// Mitsubishi GX Developer project: PLC_PCO520L2   PLC: Q06UDEH   Door Open Auto Flow

PROGRAM AT_DOAT
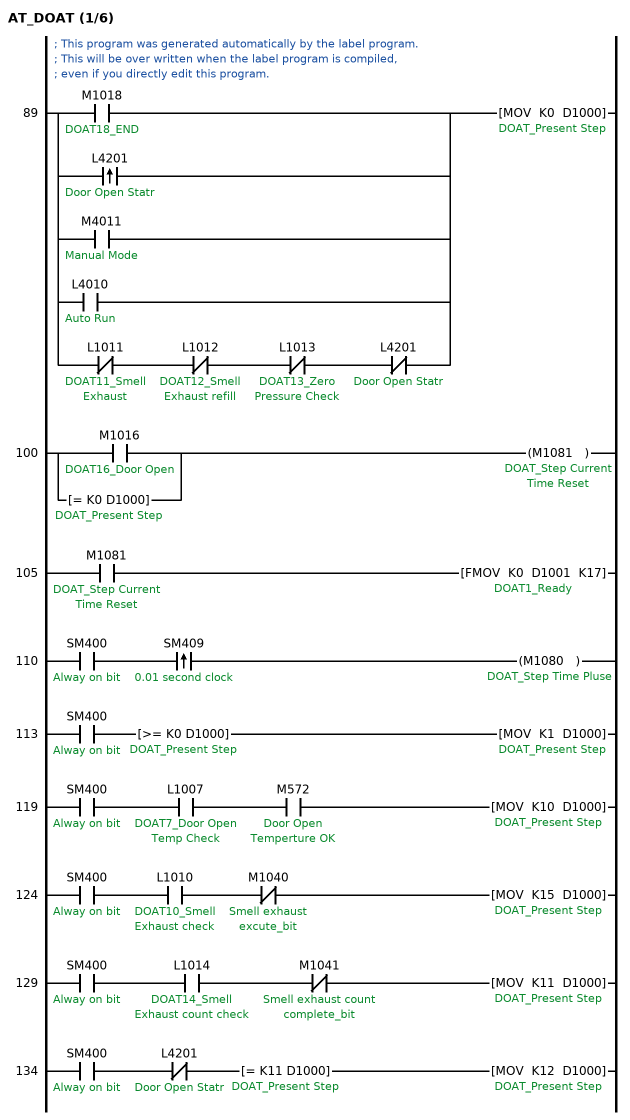
; This program was generated automatically by the label program.
; This will be over written when the label program is compiled,
; even if you directly edit this program.
89    LD      M1018  ; DOAT18_END
      ORP     L4201  ; Door Open Statr
      OR      M4011  ; Manual Mode
      OR      L4010  ; Auto Run
      LDI     L1011  ; DOAT11_Smell Exhaust
      ANI     L1012  ; DOAT12_Smell Exhaust refill
      ANI     L1013  ; DOAT13_Zero Pressure Check
      ANI     L4201  ; Door Open Statr
      ORB
      MOV     K0 D1000  ; DOAT_Present Step
100   LD      M1016  ; DOAT16_Door Open
      OR=     K0 D1000  ; DOAT_Present Step
      OUT     M1081  ; DOAT_Step Current Time Reset
105   LD      M1081  ; DOAT_Step Current Time Reset
      FMOV    K0 D1001 K17  ; DOAT1_Ready
110   LD      SM400  ; Alway on bit
      ANDP    SM409  ; 0.01 second clock
      OUT     M1080  ; DOAT_Step Time Pluse
113   LD      SM400  ; Alway on bit
      AND>=   K0 D1000  ; DOAT_Present Step
      MOV     K1 D1000
119   LD      SM400  ; Alway on bit
      AND     L1007  ; DOAT7_Door Open Temp Check
      AND     M572  ; Door Open Temperture OK
      MOV     K10 D1000
124   LD      SM400  ; Alway on bit
      AND     L1010  ; DOAT10_Smell Exhaust check
      ANI     M1040  ; Smell exhaust excute_bit
      MOV     K15 D1000
129   LD      SM400  ; Alway on bit
      AND     L1014  ; DOAT14_Smell Exhaust count check
      ANI     M1041  ; Smell exhaust count complete_bit
      MOV     K11 D1000
134   LD      SM400  ; Alway on bit
      ANI     L4201  ; Door Open Statr
      AND=    K11 D1000  ; DOAT_Present Step
      MOV     K12 D1000
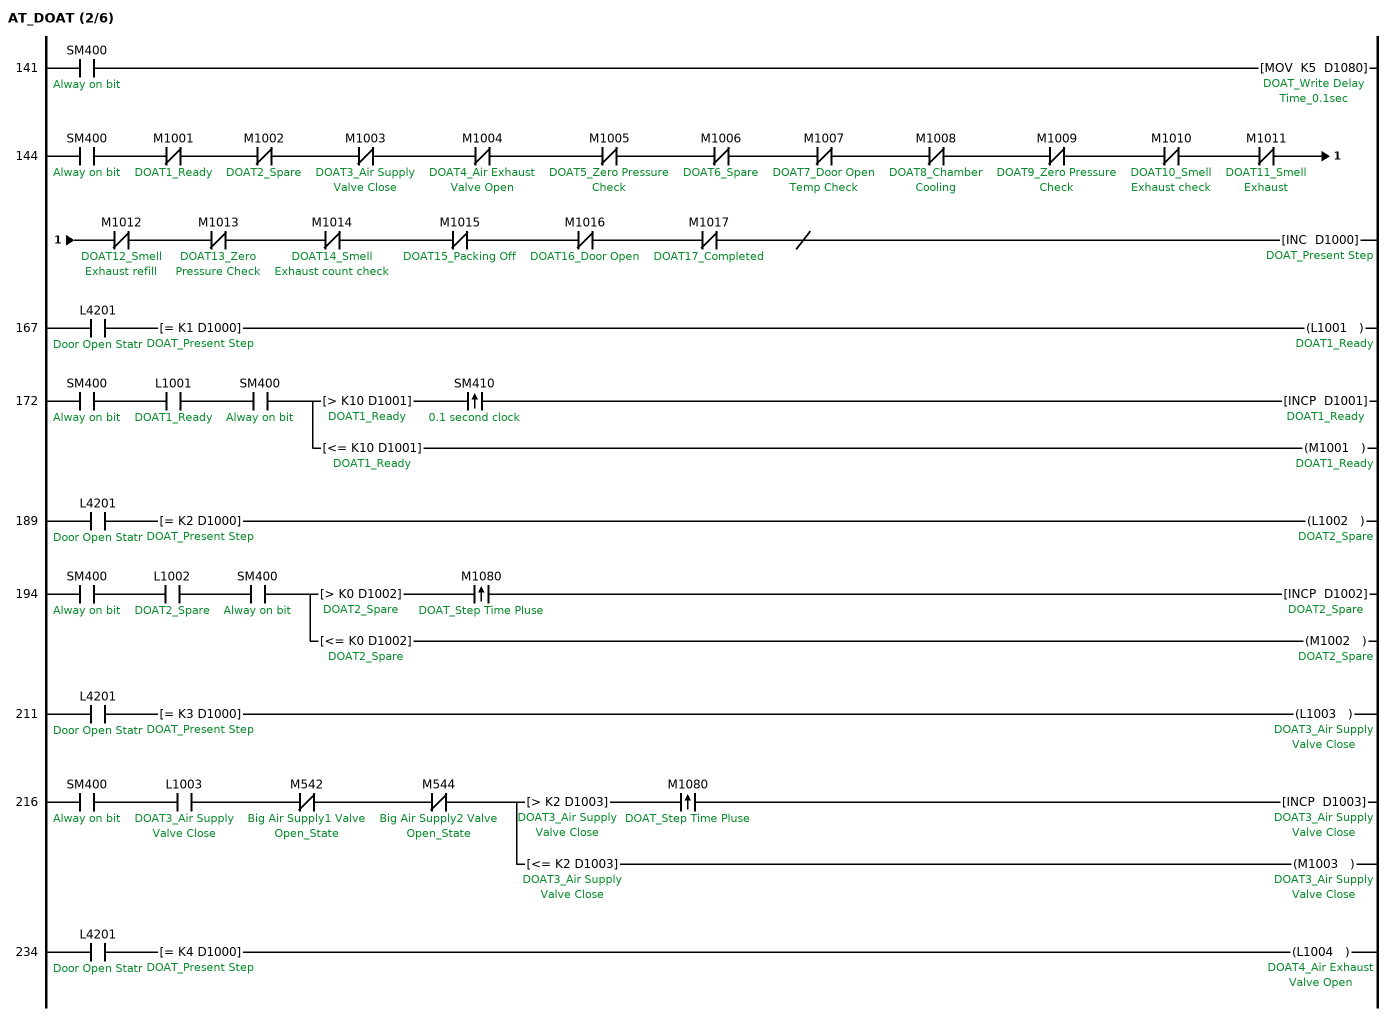
141   LD      SM400  ; Alway on bit
      MOV     K5 D1080  ; DOAT_Write Delay Time_0.1sec
144   LD      SM400  ; Alway on bit
      ANI     M1001  ; DOAT1_Ready
      ANI     M1002  ; DOAT2_Spare
      ANI     M1003  ; DOAT3_Air Supply Valve Close
      ANI     M1004  ; DOAT4_Air Exhaust Valve Open
      ANI     M1005  ; DOAT5_Zero Pressure Check
      ANI     M1006  ; DOAT6_Spare
      ANI     M1007  ; DOAT7_Door Open Temp Check
      ANI     M1008  ; DOAT8_Chamber Cooling
      ANI     M1009  ; DOAT9_Zero Pressure Check
      ANI     M1010  ; DOAT10_Smell Exhaust check
      ANI     M1011  ; DOAT11_Smell Exhaust
      ANI     M1012  ; DOAT12_Smell Exhaust refill
      ANI     M1013  ; DOAT13_Zero Pressure Check
      ANI     M1014  ; DOAT14_Smell Exhaust count check
      ANI     M1015  ; DOAT15_Packing Off
      ANI     M1016  ; DOAT16_Door Open
      ANI     M1017  ; DOAT17_Completed
      INV
      INC     D1000
; 
167   LD      L4201  ; Door Open Statr
      AND=    K1 D1000  ; DOAT_Present Step
      OUT     L1001  ; DOAT1_Ready
172   LD      SM400  ; Alway on bit
      AND     L1001  ; DOAT1_Ready
      AND     SM400  ; Alway on bit
      MPS
      AND>    K10 D1001  ; DOAT1_Ready
      ANDP    SM410  ; 0.1 second clock
      INCP    D1001
      MPP
      AND<=   K10 D1001  ; DOAT1_Ready
      OUT     M1001  ; DOAT1_Ready
; 
189   LD      L4201  ; Door Open Statr
      AND=    K2 D1000  ; DOAT_Present Step
      OUT     L1002  ; DOAT2_Spare
194   LD      SM400  ; Alway on bit
      AND     L1002  ; DOAT2_Spare
      AND     SM400  ; Alway on bit
      MPS
      AND>    K0 D1002  ; DOAT2_Spare
      ANDP    M1080  ; DOAT_Step Time Pluse
      INCP    D1002
      MPP
      AND<=   K0 D1002  ; DOAT2_Spare
      OUT     M1002  ; DOAT2_Spare
; 
211   LD      L4201  ; Door Open Statr
      AND=    K3 D1000  ; DOAT_Present Step
      OUT     L1003  ; DOAT3_Air Supply Valve Close
216   LD      SM400  ; Alway on bit
      AND     L1003  ; DOAT3_Air Supply Valve Close
      ANI     M542  ; Big Air Supply1 Valve Open_State
      ANI     M544  ; Big Air Supply2 Valve Open_State
      MPS
      AND>    K2 D1003  ; DOAT3_Air Supply Valve Close
      ANDP    M1080  ; DOAT_Step Time Pluse
      INCP    D1003
      MPP
      AND<=   K2 D1003  ; DOAT3_Air Supply Valve Close
      OUT     M1003  ; DOAT3_Air Supply Valve Close
; 
234   LD      L4201  ; Door Open Statr
      AND=    K4 D1000  ; DOAT_Present Step
      OUT     L1004  ; DOAT4_Air Exhaust Valve Open
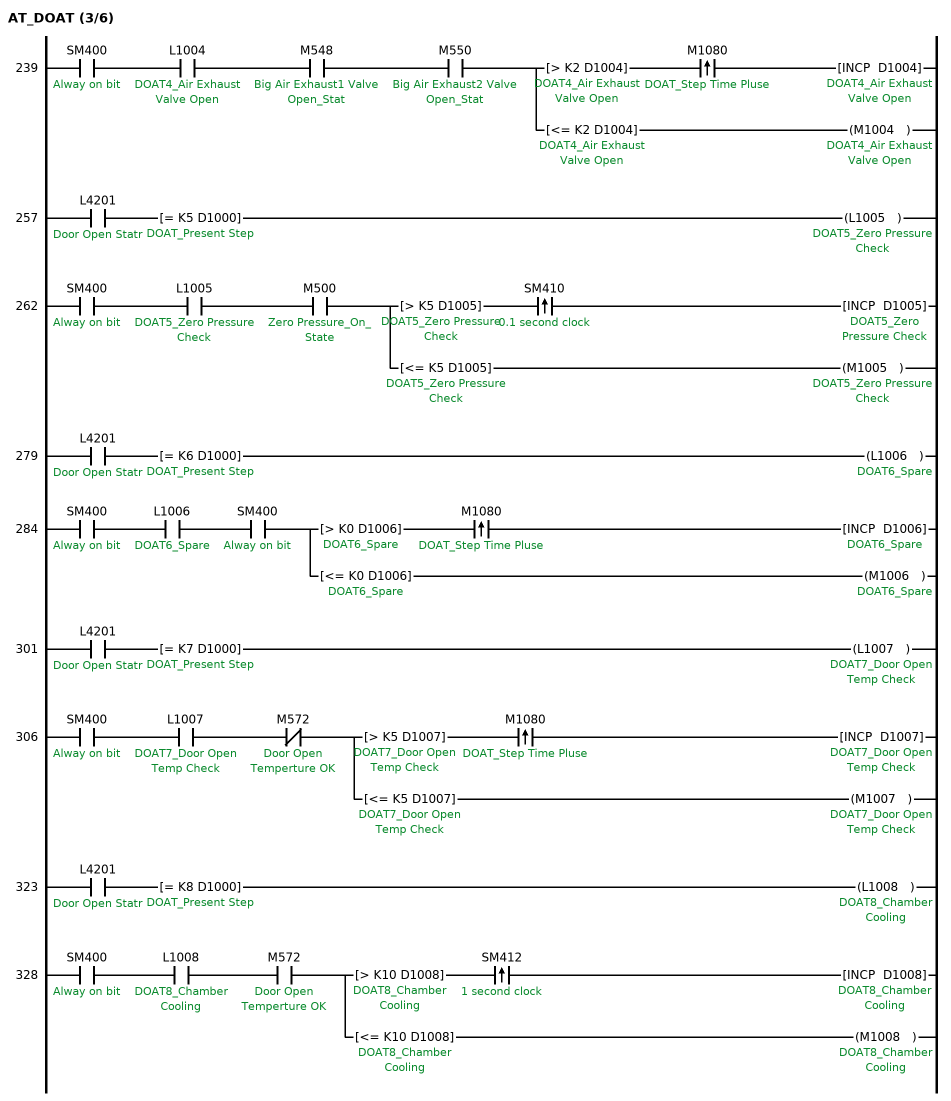
239   LD      SM400  ; Alway on bit
      AND     L1004  ; DOAT4_Air Exhaust Valve Open
      AND     M548  ; Big Air Exhaust1 Valve Open_Stat
      AND     M550  ; Big Air Exhaust2 Valve Open_Stat
      MPS
      AND>    K2 D1004  ; DOAT4_Air Exhaust Valve Open
      ANDP    M1080  ; DOAT_Step Time Pluse
      INCP    D1004
      MPP
      AND<=   K2 D1004  ; DOAT4_Air Exhaust Valve Open
      OUT     M1004  ; DOAT4_Air Exhaust Valve Open
; 
257   LD      L4201  ; Door Open Statr
      AND=    K5 D1000  ; DOAT_Present Step
      OUT     L1005  ; DOAT5_Zero Pressure Check
262   LD      SM400  ; Alway on bit
      AND     L1005  ; DOAT5_Zero Pressure Check
      AND     M500  ; Zero Pressure_On_State
      MPS
      AND>    K5 D1005  ; DOAT5_Zero Pressure Check
      ANDP    SM410  ; 0.1 second clock
      INCP    D1005
      MPP
      AND<=   K5 D1005  ; DOAT5_Zero Pressure Check
      OUT     M1005  ; DOAT5_Zero Pressure Check
; 
279   LD      L4201  ; Door Open Statr
      AND=    K6 D1000  ; DOAT_Present Step
      OUT     L1006  ; DOAT6_Spare
284   LD      SM400  ; Alway on bit
      AND     L1006  ; DOAT6_Spare
      AND     SM400  ; Alway on bit
      MPS
      AND>    K0 D1006  ; DOAT6_Spare
      ANDP    M1080  ; DOAT_Step Time Pluse
      INCP    D1006
      MPP
      AND<=   K0 D1006  ; DOAT6_Spare
      OUT     M1006  ; DOAT6_Spare
; 
301   LD      L4201  ; Door Open Statr
      AND=    K7 D1000  ; DOAT_Present Step
      OUT     L1007  ; DOAT7_Door Open Temp Check
306   LD      SM400  ; Alway on bit
      AND     L1007  ; DOAT7_Door Open Temp Check
      ANI     M572  ; Door Open Temperture OK
      MPS
      AND>    K5 D1007  ; DOAT7_Door Open Temp Check
      ANDP    M1080  ; DOAT_Step Time Pluse
      INCP    D1007
      MPP
      AND<=   K5 D1007  ; DOAT7_Door Open Temp Check
      OUT     M1007  ; DOAT7_Door Open Temp Check
; 
323   LD      L4201  ; Door Open Statr
      AND=    K8 D1000  ; DOAT_Present Step
      OUT     L1008  ; DOAT8_Chamber Cooling
328   LD      SM400  ; Alway on bit
      AND     L1008  ; DOAT8_Chamber Cooling
      AND     M572  ; Door Open Temperture OK
      MPS
      AND>    K10 D1008  ; DOAT8_Chamber Cooling
      ANDP    SM412  ; 1 second clock
      INCP    D1008
      MPP
      AND<=   K10 D1008  ; DOAT8_Chamber Cooling
      OUT     M1008  ; DOAT8_Chamber Cooling
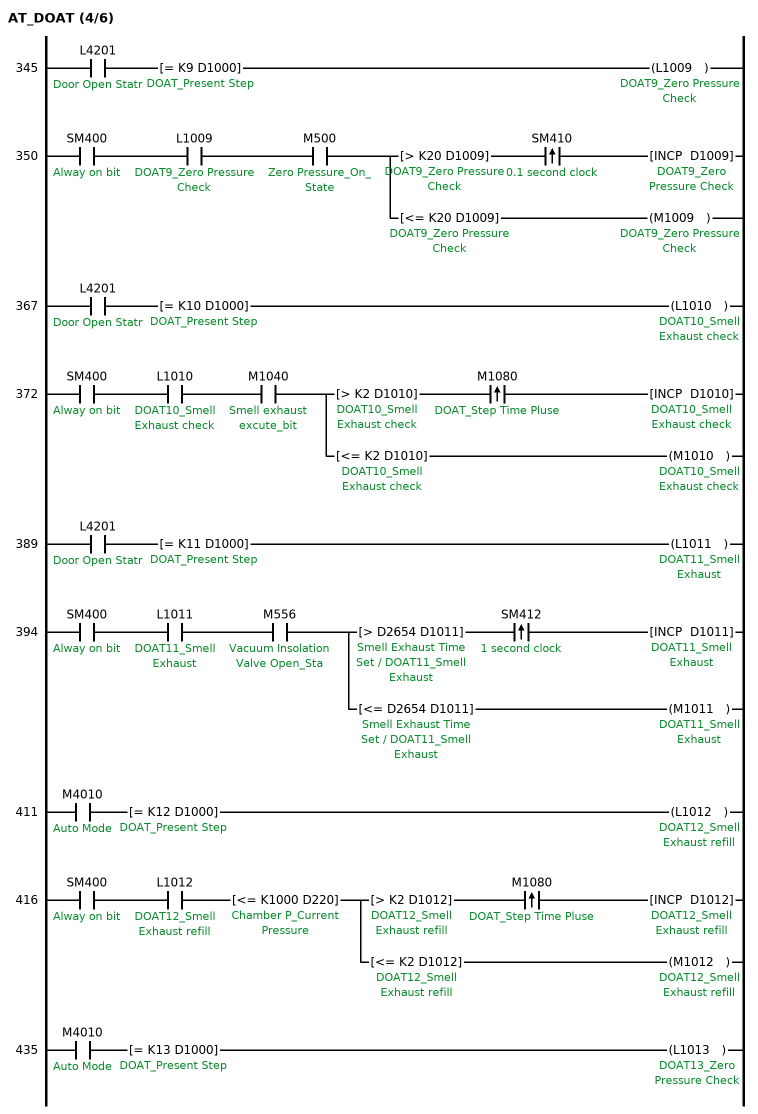
; 
345   LD      L4201  ; Door Open Statr
      AND=    K9 D1000  ; DOAT_Present Step
      OUT     L1009  ; DOAT9_Zero Pressure Check
350   LD      SM400  ; Alway on bit
      AND     L1009  ; DOAT9_Zero Pressure Check
      AND     M500  ; Zero Pressure_On_State
      MPS
      AND>    K20 D1009  ; DOAT9_Zero Pressure Check
      ANDP    SM410  ; 0.1 second clock
      INCP    D1009
      MPP
      AND<=   K20 D1009  ; DOAT9_Zero Pressure Check
      OUT     M1009  ; DOAT9_Zero Pressure Check
; 
367   LD      L4201  ; Door Open Statr
      AND=    K10 D1000  ; DOAT_Present Step
      OUT     L1010  ; DOAT10_Smell Exhaust check
372   LD      SM400  ; Alway on bit
      AND     L1010  ; DOAT10_Smell Exhaust check
      AND     M1040  ; Smell exhaust excute_bit
      MPS
      AND>    K2 D1010  ; DOAT10_Smell Exhaust check
      ANDP    M1080  ; DOAT_Step Time Pluse
      INCP    D1010
      MPP
      AND<=   K2 D1010  ; DOAT10_Smell Exhaust check
      OUT     M1010  ; DOAT10_Smell Exhaust check
; 
389   LD      L4201  ; Door Open Statr
      AND=    K11 D1000  ; DOAT_Present Step
      OUT     L1011  ; DOAT11_Smell Exhaust
394   LD      SM400  ; Alway on bit
      AND     L1011  ; DOAT11_Smell Exhaust
      AND     M556  ; Vacuum Insolation Valve Open_Sta
      MPS
      AND>    D2654 D1011  ; Smell Exhaust Time Set / DOAT11_Smell Exhaust
      ANDP    SM412  ; 1 second clock
      INCP    D1011
      MPP
      AND<=   D2654 D1011  ; Smell Exhaust Time Set / DOAT11_Smell Exhaust
      OUT     M1011  ; DOAT11_Smell Exhaust
; 
411   LD      M4010  ; Auto Mode
      AND=    K12 D1000  ; DOAT_Present Step
      OUT     L1012  ; DOAT12_Smell Exhaust refill
416   LD      SM400  ; Alway on bit
      AND     L1012  ; DOAT12_Smell Exhaust refill
      AND<=   K1000 D220  ; Chamber P_Current Pressure
      MPS
      AND>    K2 D1012  ; DOAT12_Smell Exhaust refill
      ANDP    M1080  ; DOAT_Step Time Pluse
      INCP    D1012
      MPP
      AND<=   K2 D1012  ; DOAT12_Smell Exhaust refill
      OUT     M1012  ; DOAT12_Smell Exhaust refill
; 
435   LD      M4010  ; Auto Mode
      AND=    K13 D1000  ; DOAT_Present Step
      OUT     L1013  ; DOAT13_Zero Pressure Check
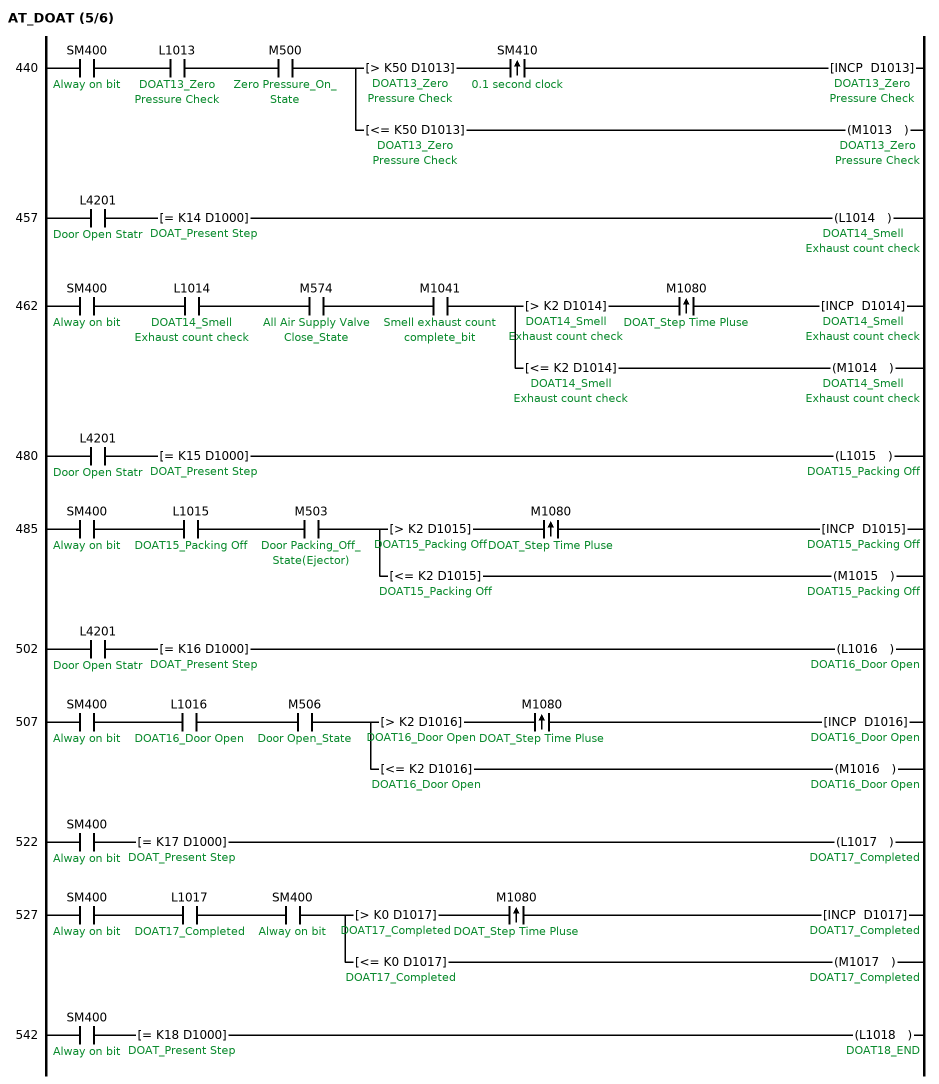
440   LD      SM400  ; Alway on bit
      AND     L1013  ; DOAT13_Zero Pressure Check
      AND     M500  ; Zero Pressure_On_State
      MPS
      AND>    K50 D1013  ; DOAT13_Zero Pressure Check
      ANDP    SM410  ; 0.1 second clock
      INCP    D1013
      MPP
      AND<=   K50 D1013  ; DOAT13_Zero Pressure Check
      OUT     M1013  ; DOAT13_Zero Pressure Check
; 
457   LD      L4201  ; Door Open Statr
      AND=    K14 D1000  ; DOAT_Present Step
      OUT     L1014  ; DOAT14_Smell Exhaust count check
462   LD      SM400  ; Alway on bit
      AND     L1014  ; DOAT14_Smell Exhaust count check
      AND     M574  ; All Air Supply Valve Close_State
      AND     M1041  ; Smell exhaust count complete_bit
      MPS
      AND>    K2 D1014  ; DOAT14_Smell Exhaust count check
      ANDP    M1080  ; DOAT_Step Time Pluse
      INCP    D1014
      MPP
      AND<=   K2 D1014  ; DOAT14_Smell Exhaust count check
      OUT     M1014  ; DOAT14_Smell Exhaust count check
; 
480   LD      L4201  ; Door Open Statr
      AND=    K15 D1000  ; DOAT_Present Step
      OUT     L1015  ; DOAT15_Packing Off
485   LD      SM400  ; Alway on bit
      AND     L1015  ; DOAT15_Packing Off
      AND     M503  ; Door Packing_Off_State(Ejector)
      MPS
      AND>    K2 D1015  ; DOAT15_Packing Off
      ANDP    M1080  ; DOAT_Step Time Pluse
      INCP    D1015
      MPP
      AND<=   K2 D1015  ; DOAT15_Packing Off
      OUT     M1015  ; DOAT15_Packing Off
; 
502   LD      L4201  ; Door Open Statr
      AND=    K16 D1000  ; DOAT_Present Step
      OUT     L1016  ; DOAT16_Door Open
507   LD      SM400  ; Alway on bit
      AND     L1016  ; DOAT16_Door Open
      AND     M506  ; Door Open_State
      MPS
      AND>    K2 D1016  ; DOAT16_Door Open
      ANDP    M1080  ; DOAT_Step Time Pluse
      INCP    D1016
      MPP
      AND<=   K2 D1016  ; DOAT16_Door Open
      OUT     M1016  ; DOAT16_Door Open
522   LD      SM400  ; Alway on bit
      AND=    K17 D1000  ; DOAT_Present Step
      OUT     L1017  ; DOAT17_Completed
527   LD      SM400  ; Alway on bit
      AND     L1017  ; DOAT17_Completed
      AND     SM400  ; Alway on bit
      MPS
      AND>    K0 D1017  ; DOAT17_Completed
      ANDP    M1080  ; DOAT_Step Time Pluse
      INCP    D1017
      MPP
      AND<=   K0 D1017  ; DOAT17_Completed
      OUT     M1017  ; DOAT17_Completed
542   LD      SM400  ; Alway on bit
      AND=    K18 D1000  ; DOAT_Present Step
      OUT     L1018  ; DOAT18_END
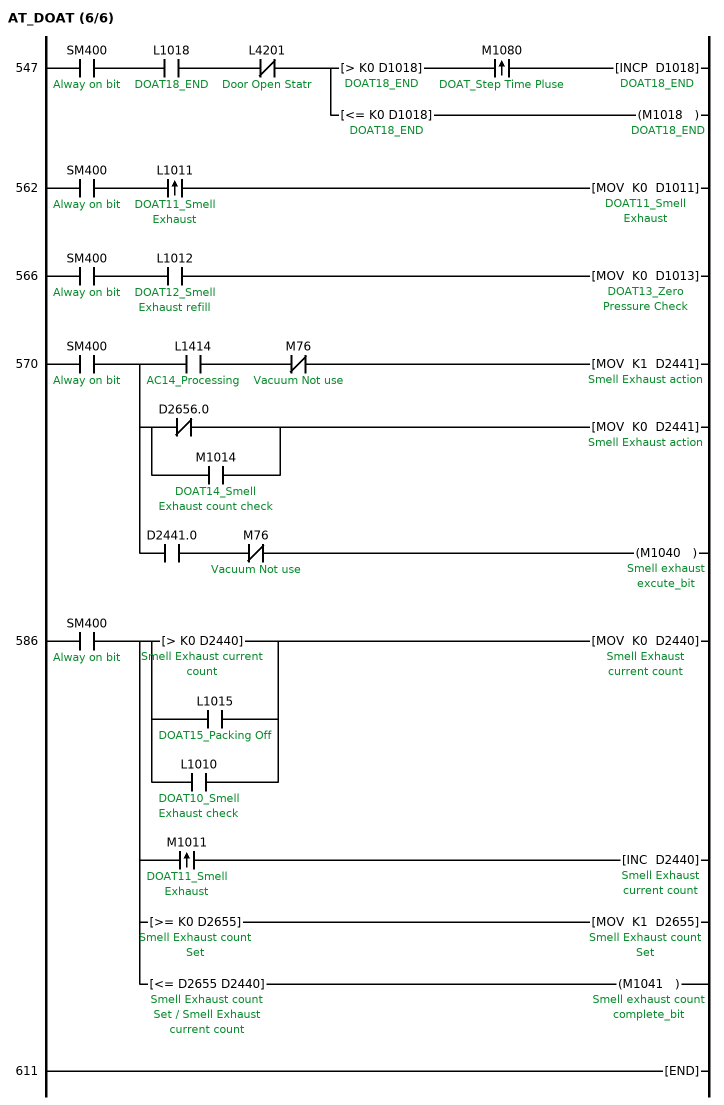
547   LD      SM400  ; Alway on bit
      AND     L1018  ; DOAT18_END
      ANI     L4201  ; Door Open Statr
      MPS
      AND>    K0 D1018  ; DOAT18_END
      ANDP    M1080  ; DOAT_Step Time Pluse
      INCP    D1018
      MPP
      AND<=   K0 D1018  ; DOAT18_END
      OUT     M1018  ; DOAT18_END
562   LD      SM400  ; Alway on bit
      ANDP    L1011  ; DOAT11_Smell Exhaust
      MOV     K0 D1011
566   LD      SM400  ; Alway on bit
      AND     L1012  ; DOAT12_Smell Exhaust refill
      MOV     K0 D1013
570   LD      SM400  ; Alway on bit
      MPS
      AND     L1414  ; AC14_Processing
      ANI     M76  ; Vacuum Not use
      MOV     K1 D2441  ; Smell Exhaust action
      MRD
      LDI     D2656.0
      OR      M1014  ; DOAT14_Smell Exhaust count check
      ANB
      MOV     K0 D2441
      MPP
      AND     D2441.0
      ANI     M76  ; Vacuum Not use
      OUT     M1040  ; Smell exhaust excute_bit
586   LD      SM400  ; Alway on bit
      MPS
      LD>     K0 D2440  ; Smell Exhaust current count
      OR      L1015  ; DOAT15_Packing Off
      OR      L1010  ; DOAT10_Smell Exhaust check
      ANB
      MOV     K0 D2440
      MRD
      ANDP    M1011  ; DOAT11_Smell Exhaust
      INC     D2440
      MRD
      AND>=   K0 D2655  ; Smell Exhaust count Set
      MOV     K1 D2655
      MPP
      AND<=   D2655 D2440  ; Smell Exhaust count Set / Smell Exhaust current count
      OUT     M1041  ; Smell exhaust count complete_bit
611   END
END_PROGRAM
